// TIA Portal V17 export
// export: Created 2024-09-02T12:50:25.856982Z, ExportSetting WithDefaults, DisplayName Totally Integrated Automation Portal, DisplayVersion V17, DisplayName TIA Portal Openness, DisplayVersion V17, DisplayName TIA Portal Version Control Interface, DisplayVersion V17, DisplayName STEP 7 Professional, DisplayVersion V17, DisplayName STEP 7 Safety, DisplayVersion V17, DisplayName WinCC Professional, DisplayVersion V17
VAR_GLOBAL   // PLC tag table "OP70_2"
   IW_RFID_SLG3_OP70_3 AT %IW2004 : Word;   // Balluff BIS V Reader 2 (+M01-BX602)
   I_MM150_Z_Axis_Gripper_UP_OP70_2 AT %I54.0 : Bool;
   I_MM150_Z_Axis_Gripper_Down_OP70_2 AT %I54.1 : Bool;
   I_MM160_Z_Axis_Screwdrive_UP_OP70_2 AT %I54.2 : Bool;
   I_MM160_Z_Axis_Screwdrive_Down_OP70_2 AT %I54.3 : Bool;
   I_MM170_Z_Axis_Screwdrive_Unit_UP_OP70_2 AT %I54.4 : Bool;
   I_MM170_Z_Axis_Screwdrive_Unit_Down_OP70_2 AT %I54.5 : Bool;
   I_MM180_Z_Axis_Screwdrive_Unit_Clamps_Open_OP70_2 AT %I54.6 : Bool;
   I_Safety_bolt_Z_Axis_Screwdrive AT %I54.7 : Bool;
   I_Presure_on_Gripper_OK AT %I53.7 : Bool;
   I_MM130_Press_Damper_Down_OP70_2 AT %I53.4 : Bool;
   I_MM140_Y_Axis_Gripper_Back_OP70_2 AT %I53.5 : Bool;
   I_MM50_index_Camera_Down_OP70_2 AT %I51.2 : Bool;
   I_MM50_index_Camera_Up_OP70_2 AT %I51.3 : Bool;
   I_MM51_index_Camera_Down_OP70_2 AT %I51.4 : Bool;
   I_MM51_index_Camera_Up_OP70_2 AT %I51.5 : Bool;
   I_MM60_Stopper_Screwdriver_Close_OP70_2 AT %I51.6 : Bool;
   I_MM60_pallet_at_Stopper_Screwdriver_OP70_2 AT %I51.7 : Bool;
   "I_MM70/71_index_Screwdriver_Down_OP70_2" AT %I52.0 : Bool;
   "I_MM70/71_index_Screwdriver_UP_OP70_2" AT %I52.1 : Bool;
   I_Pallet_at_Outlet_Station AT %I52.2 : Bool;
   I_MM40_Stopper_Camera_Close_OP70_2 AT %I50.4 : Bool;
   I_MM40_pallet_at_Stopper_Camera_OP70_2 AT %I50.5 : Bool;
   Q_Vacuum_Gripper_Drop_Pulse_OP70_2 AT %Q2.1 : Bool;
   Q_Vacuum_Gripper_ON_OP70_2 AT %Q2.2 : Bool;
   Q_Camera_Light_ON_OP70_2 AT %Q2.3 : Bool;
   Q_MM40_Stopper_Camera_Open_Camera_OP70_2 AT %Q81.2 : Bool;
   "Q_MM50/51_index_Camera_Upward_OP70_2" AT %Q82.0 : Bool;
   "Q_MM50/51_index_Camera_Downward_OP70_2" AT %Q82.1 : Bool;
   Q_MM60_Stopper_Screwdriver_Open_OP70_2 AT %Q82.2 : Bool;
   "Q_MM70/71_index_Screwdriver_Upward_OP70_2" AT %Q83.0 : Bool;
   "Q_MM70/71_index_Screwdriver_Downward_OP70_2" AT %Q83.1 : Bool;
   Q_MM140_Y_Axis_Gripper_Forward_OP70_2 AT %Q87.2 : Bool;
   Q_MM140_Y_Axis_Gripper_Backward_OP70_2 AT %Q87.3 : Bool;
   Q_MM150_Z_Axis_Gripper_Downward_OP70_2 AT %Q88.0 : Bool;
   Q_MM150_Z_Axis_Gripper_Upward_OP70_2 AT %Q88.1 : Bool;
   Q_MM160_Z_Axis_Screwdrive_Downward_OP70_2 AT %Q88.2 : Bool;
   Q_MM160_Z_Axis_Screwdrive_Upward_OP70_2 AT %Q88.3 : Bool;
   Q_MM170_Z_Axis_Screwdrive_Unit_Downward_OP70_2 AT %Q89.0 : Bool;
   Q_MM170_Z_Axis_Screwdrive_Unit_Upward_OP70_2 AT %Q89.1 : Bool;
   Q_MM180_Z_Axis_Screwdrive_Unit_Clamps_Open_OP70_2 AT %Q89.2 : Bool;
   QW_RFID_SLG3_OP70_3 AT %QW2004 : Word;   // Balluff BIS V Reader 1 (+M01-BX600)
   Q_MM190_Z_Axis_Screwdrive_Unit_Clamps_2_Open_OP70_2 AT %Q90.0 : Bool;
   IW_RFID_SLG2_OP70_2 AT %IW2102 : Word;   // Balluff BIS V Reader 1 (+M01-BX600)
   QW_RFID_SLG2_OP70_2 AT %QW2102 : Word;   // Balluff BIS V Reader 1 (+M01-BX600)
   I_Pressure_on_clamping_OK AT %I52.3 : Bool;
   I_Ball_Controle_Present AT %I56.7 : Bool;
END_VAR
